// TIA Portal project "Test_Zeiten" (V20)

(* hardware
DEVICE "S7-300/ET200M-Station_1"  S7-300 station
   slot 0: "Profilschiene_0"  Rail  6ES7 390-1***0-0AA0
   slot 2: "PLC_1"  CPU 315-2 PN/DP  6ES7 315-2EH14-0AB0  V3.2.18
      slot 2: "PROFINET-Schnittstelle_1"  PN-IO
         slot 1: "Port_1"  Port
         slot 2: "Port_2"  Port
   slot 4: "DI 16x24VDC_1"  DI16 x 24VDC, interrupt  6ES7 321-7BH01-0AB0
   slot 5: "DO 8x24VDC/0.5A_1"  DO8 x 24VDC / 0.5A  6ES7 322-8BF00-0AB0
*)

// ===== PLC "PLC_1"  CPU 315-2 PN/DP =====

VAR_GLOBAL   // PLC tag table "Standard-Variablentabelle"
   "M1" AT %A0.0 : Bool;
   "M2" AT %A0.1 : Bool;
   "M3" AT %A0.2 : Bool;
   "S1" AT %E0.0 : Bool;   // Not-Aus
   "S2" AT %E0.1 : Bool;   // Start-Taster
   "Tag_1" AT %M1.0 : Bool;
END_VAR

FUNCTION "Zeiten_Test" : Void   // FC1, FBD
{ S7_Optimized_Access := 'FALSE' }
VERSION : 0.1
BEGIN

REGION Network 1: Impuls
   // Der Impuls hält ein Signal nur so lange aktiv, bis die Zeit abgelaufen ist. Danach gibt er das Signal mehr nicht weiter.
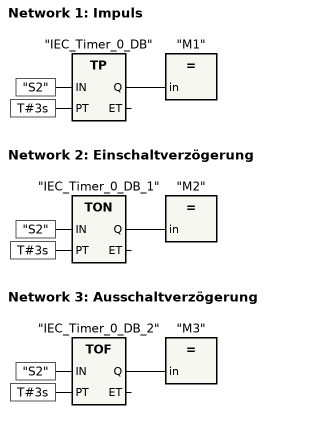
   "IEC_Timer_0_DB".TP(IN := "S2", PT := T#3s);
   "M1" := "IEC_Timer_0_DB".Q;
END_REGION

REGION Network 2: Einschaltverzögerung
   // Die Einschaltverzögerung gibt das Signal erst weiter, wenn die Zeit abgelaufen ist. Danach gibt Sie das Signal unbegrenzt lange weiter.
   "IEC_Timer_0_DB_1".TON(IN := "S2", PT := T#3s);
   "M2" := "IEC_Timer_0_DB_1".Q;
END_REGION

REGION Network 3: Ausschaltverzögerung
   // Die Ausschaltverzögerung gibt das Signal unbegrenzt lange weiter und hält es so lange aktiv, bis die Zeit abgelaufen ist.
   "IEC_Timer_0_DB_2".TOF(IN := "S2", PT := T#3s);
   "M3" := "IEC_Timer_0_DB_2".Q;
END_REGION
END_FUNCTION

ORGANIZATION_BLOCK "Main"   // OB1, FBD
TITLE = "Main Program Sweep (Cycle)"
{ S7_Optimized_Access := 'FALSE' }
VERSION : 0.1
   VAR_TEMP
      OB1_EV_CLASS : Byte;   // Bits 0-3 = 1 (Coming event), Bits 4-7 = 1 (Event class 1)
      OB1_SCAN_1 : Byte;   // 1 (Cold restart scan 1 of OB 1), 3 (Scan 2-n of OB 1)
      OB1_PRIORITY : Byte;   // Priority of OB Execution
      OB1_OB_NUMBR : Byte;   // 1 (Organization block 1, OB1)
      OB1_RESERVED_1 : Byte;   // Reserved for system
      OB1_RESERVED_2 : Byte;   // Reserved for system
      OB1_PREV_CYCLE : Int;   // Cycle time of previous OB1 scan (milliseconds)
      OB1_MIN_CYCLE : Int;   // Minimum cycle time of OB1 (milliseconds)
      OB1_MAX_CYCLE : Int;   // Maximum cycle time of OB1 (milliseconds)
      OB1_DATE_TIME : Date_And_Time;   // Date and time OB1 started
   END_VAR
BEGIN

REGION Network 1
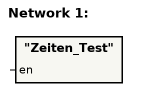
   "Zeiten_Test"();
END_REGION
END_ORGANIZATION_BLOCK